{attribute 'qualified_only'}
{attribute 'strict'}
TYPE E_Message_EM :
(
	eNoMessage := 0,
	eTooMuchElectricMeter := 1,
	eElectricMeterError := 2,
	eNoConnectionToBackend := 3,
	eElectricMeterWarning :=4
);
END_TYPE

(* stored: Version 1.1.0.1, ProductVersion 3.1.4024.9
   DUT E_Message_EM: Id {54f0f5a3-52d2-426a-abc0-0cc03134eb8c} *)
